PROGRAM Cell_Sequencer
VAR
END_VAR

CASE Cell.StateManager.oState OF
	State.Aborting:		Cell_SeqAborting();
	State.Aborted:		Cell_SeqAborted();
	State.Resetting:	Cell_SeqResetting();
	State.Stopped:		Cell_SeqStopped();
	State.Starting:		Cell_SeqStarting();
	State.Running:		Cell_SeqRunning();
	State.Pausing:		Cell_SeqPausing();
	State.Paused:		Cell_SeqPaused();
	State.Resuming:		Cell_SeqResuming();
	State.Stopping:		Cell_SeqStopping();	
END_CASE

ACTION Cell_SeqAborted:

END_ACTION

ACTION Cell_SeqAborting:
Comp01.StateManager.iCmd := Cmd.Abort;
//Comp02.StateManager.iCmd := Cmd.Abort;

IF Comp01.StateManager.oState = State.Aborted THEN //AND Comp02.StateManager.oState = State.Aborted THEN
	Cell.StateManager.iSeqComplete := TRUE;
END_IF
END_ACTION

ACTION Cell_SeqPaused:

END_ACTION

ACTION Cell_SeqPausing:
Comp01.StateManager.iCmd := Cmd.Pause;
//Comp02.StateManager.iCmd := Cmd.Pause;

IF Comp01.StateManager.oState = State.Paused THEN //AND Comp02.StateManager.oState = State.Paused THEN
	Cell.StateManager.iSeqComplete := TRUE;
END_IF
END_ACTION

ACTION Cell_SeqResetting:
Comp01.StateManager.iCmd := Cmd.Reset;
//Comp02.StateManager.iCmd := Cmd.Reset;

IF Comp01.StateManager.oState = State.Stopped THEN //AND Comp02.StateManager.oState = State.Stopped THEN
	Cell.StateManager.iSeqComplete := TRUE;
END_IF
END_ACTION

ACTION Cell_SeqResuming:
Comp01.StateManager.iCmd := Cmd.Resume;
//Comp02.StateManager.iCmd := Cmd.Resume;

IF Comp01.StateManager.oState = State.Running THEN //AND Comp02.StateManager.oState = State.Running THEN
	Cell.StateManager.iSeqComplete := TRUE;
END_IF
END_ACTION

ACTION Cell_SeqRunning:


IF Comp01.StateManager.oState = State.Stopping THEN //AND Comp02.StateManager.oState = State.Stopping THEN
	Cell.StateManager.iSeqComplete := TRUE;
END_IF
END_ACTION

ACTION Cell_SeqStarting:
Comp01.StateManager.iCmd := Cmd.Start;
//Comp02.StateManager.iCmd := Cmd.Start;

IF Comp01.StateManager.oState = State.Running THEN //AND Comp02.StateManager.oState = State.Running THEN
	Cell.StateManager.iSeqComplete := TRUE;
END_IF
END_ACTION

ACTION Cell_SeqStopped:

END_ACTION

ACTION Cell_SeqStopping:
Comp01.StateManager.iCmd := Cmd.Stop;
//Comp02.StateManager.iCmd := Cmd.Stop;

IF Comp01.StateManager.oState = State.Stopped THEN //AND Comp02.StateManager.oState = State.Stopped THEN
	Cell.StateManager.iSeqComplete := TRUE;
END_IF
END_ACTION

END_PROGRAM

(* stored: Version 1.1.0.1, ProductVersion 3.1.4022.11
   POU Cell_Sequencer: Id {b274889a-b419-4de0-bd8f-0e93f4ab20b1}, SpecialFunc None
   Action Cell_SeqAborted: Id {9fd418e9-5b2a-4515-919b-4bd0e6a4791e}
   Action Cell_SeqAborting: Id {c646c587-e165-4123-9090-069c6b0b1d4e}
   Action Cell_SeqPaused: Id {a9ddab99-e90a-4ac7-ac2a-601735449271}
   Action Cell_SeqPausing: Id {3a69313e-d916-45cb-ada0-f3af761f234b}
   Action Cell_SeqResetting: Id {83eb45b8-dc57-4728-9b68-19f3f8bc18a0}
   Action Cell_SeqResuming: Id {07d683f3-d94d-4d11-a369-58d015755d22}
   Action Cell_SeqRunning: Id {61c1c92a-a883-4bef-b9b8-e0c7c414df08}
   Action Cell_SeqStarting: Id {796ae151-ee64-49e1-b89c-fb5108207a51}
   Action Cell_SeqStopped: Id {0da1b50b-a30a-4fb4-8c33-284d5e2b6343}
   Action Cell_SeqStopping: Id {45168a9f-26a3-429f-84ed-356293d040f6} *)
